PROGRAM Module1Control
VAR
	//Cyl1
	FB_Cylinder_Right: FB_Cylinder;
	ExtendCyl_Right: BOOL;
	Cyl_RightStatus: BOOL;
	
	//Poti 
	Poti_Scale: FB_ScaleAnalogInput;
	Poti_in AT %I* : DINT;
	{attribute 'OPC.UA.DA' := '1'}
	{attribute 'TcAnalytics'}
	Display AT %Q*:INT;
	
	
	
	FB_Cylinder_Left: FB_Cylinder;
	ExtendCyl_Left: BOOL;
	Cyl_LeftStatus: BOOL;
END_VAR

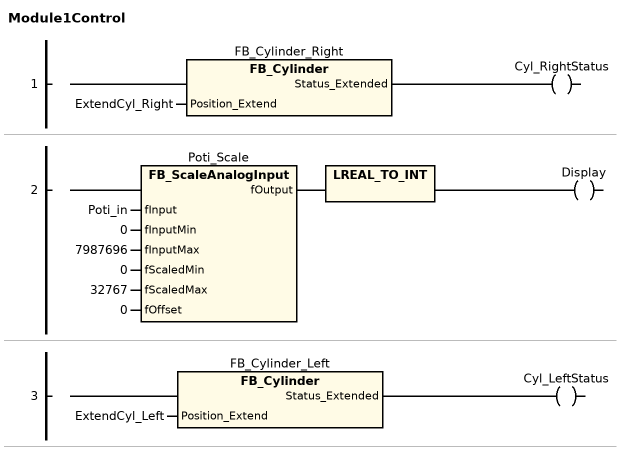
// NETWORK 1
FB_Cylinder_Right(Position_Extend := ExtendCyl_Right); // FB_Cylinder
Cyl_RightStatus := FB_Cylinder_Right.Status_Extended;

// NETWORK 2
Poti_Scale(
    fInput := Poti_in,
    fInputMin := 0,
    fInputMax := 7987696,
    fScaledMin := 0,
    fScaledMax := 32767,
    fOffset := 0); // FB_ScaleAnalogInput
Display := LREAL_TO_INT(Poti_Scale.fOutput);

// NETWORK 3
FB_Cylinder_Left(Position_Extend := ExtendCyl_Left); // FB_Cylinder
Cyl_LeftStatus := FB_Cylinder_Left.Status_Extended;

END_PROGRAM

(* stored: Version 1.1.0.1, ProductVersion 3.1.4024.4
   POU Module1Control: Id {7b30ff92-62c8-4f3a-94ee-38a451ec7199}, SpecialFunc None *)
